(* Logix 5000 project; controller Lab1 vendor 1 type 14 code 150 rev 37.11; software revision 37.00 *)

TASK MainTask (continuous, watchdog 500 ms) : MainProgram

MODULES
   Local : vendor 1 type 14 code 150 (Compact 0, rev 37.11)
      Discrete_IO : Embedded (Compact 1, rev 3.1, Output RPI 20 ms)
      Analog_IO : Embedded (Compact 2, rev 1.1, Output RPI 80 ms)
      Counters : Embedded (Compact 3, rev 1.1, Output RPI 20 ms)
END_MODULES

VAR_GLOBAL   (* controller tags *)
   ClosingDrain : STRING;
   CountDownSec : DINT;
   CountDownStr : STRING := '0';
   Countfor60cm : DINT := 30818;
   CurrentFillTarge_cm : REAL;
   CurrentMixTime_ms : DINT;
   CurrentPassVolume_mL : REAL;
   DefaultK_factor : REAL := 13190.0;
   Done_btn : ALIAS FOR Local:1:I.Data.1;
   DotStr : STRING := '.';
   DotZeroStr : STRING := '.0';
   Drain_btn : ALIAS FOR Local:1:I.Data.3;
   DrainDisplay_EU : REAL;
   DrainEU_Int : DINT;
   DrainEU_Str : STRING;
   DrainValve : ALIAS FOR Local:1:O.Data.10;
   Dump_btn : ALIAS FOR Local:1:I.Data.12;
   DumpEmpty_cm : REAL := 1.0;
   e : STRING;
   EmergencytimeCountdown : DINT;
   FillCM_Int : DINT;
   FillCM_Str : STRING;
   FillHeight_cm_HSC : REAL;
   FillSetPoint_cm : REAL := 30.0;
   Full : DINT := 29000;
   Full_Btn : ALIAS FOR Local:1:I.Data.15;
   Good_btn : ALIAS FOR Local:1:I.Data.0;
   Half : DINT := -128;
   Half_Btn : ALIAS FOR Local:1:I.Data.14;
   HSC1_CurrentCount : ALIAS FOR Local:3:I.Ctr0CurrentCount;
   HSC_Enable : ALIAS FOR Local:3:O.Ctr0En;
   HSC_ResetPulse : ALIAS FOR Local:3:O.Ctr0SoftPreset;
   HSCStr : STRING := '30818';
   InitDone : DINT;
   InitDoneAlready : DINT;
   K_factor : REAL := 12630.327;
   LevelMax : DINT := 12354;
   LevelMin : DINT := -30607;
   LevelRaw_0cm : DINT;
   LevelRaw_85cm : DINT;
   M_DrainClose1 : STRING := 'Pass 1 : Waiting for drain valve to close';
   M_DrainClose2 : STRING := 'Pass 2 : waiting for drain valve to close';
   M_DrainClose3 : STRING;
   M_Dump : STRING := 'Normal Dump. DP display EU =';
   M_EmerDraining : STRING;
   M_Emerg : STRING := 'Emergency Stop Pressed : Press Drain to empty and recover';
   M_EmergDraining : STRING := 'Emergency Draining, Seconds left';
   M_Emergencytime : STRING;
   M_Fill : STRING := 'Normal Fill : Estimated level from HSC = ';
   M_Idle : STRING := 'Proving Selected. Press Prove to begin or Zero to reset HSC';
   M_Kcalculated : STRING := 'K - Factor Calculated. Press Done to return to Waiting.';
   M_KCalculating : STRING := 'Calculating K-Factor from captured proving run..';
   M_Mix1 : STRING := 'Pass 1 Mixing for 3 seconds';
   M_Mix2 : STRING := 'Pass 2 mixing for 2 seconds';
   M_Mix3 : STRING := 'Pass 3 mixing for 5 seconds. Price = ';
   M_Pass1Dump : STRING;
   M_Pass1Fill : STRING := 'Pass 1 filling to 30cm. Height cm =';
   M_Pass2 : STRING := 'Pass 2 preparation: resetting HSC and loading second targer';
   M_Pass2Dump : STRING := 'Pass 2 dumping. Batch finishing';
   M_Pass2Fill : STRING := 'Pass 2 filling to 20 cm. Height cm = ';
   M_Pass3Dump : STRING := 'Pass 3 dumping. Final Price = ';
   M_Pass3Fill : STRING := 'Pass 3 Filling to 50 cm. Height = ';
   M_price : STRING := '   Price in dollars = ';
   M_Proving : STRING := 'Proving: Fill. Press Good @ 60 cm , HSC  = ';
   M_Proving_Closing : STRING := 'Proving: Waiting for drain to close. Second left =';
   M_Proving_Starting : STRING := 'Proving setup: capturing low level and closing drain.';
   M_RevDrainClose1 : STRING := 'Reverse Drain Closing 1';
   M_RevDrainClose2 : STRING := 'Reverse Drain Closing 2';
   M_RevDump1 : STRING := 'Reverse Dump 1 EU';
   M_RevDump2 : STRING := 'Reverse Dump 2 EU';
   M_RevFill1 : STRING := 'Reverse Fill 1 cm';
   M_RevFill2 : STRING := 'Reverse Fill 2 cm';
   M_RevMix1 : STRING := 'Reverse Mix 1';
   M_RevMix2 : STRING := 'Reverse Mix 2';
   m_state3 : STRING;
   M_StopDump : STRING := 'Stop Dump actice. DP Display EU = ';
   M_StopHold : STRING := 'Stopped. Press Dump to empty tank and reset displayed volume.';
   M_TotalmL : STRING := 'Total Volume mL = ';
   M_Waiting2 : STRING := 'Waiting: Press Start, Reverse, or Prove';
   MaxTime_ms : DINT;
   Mixer : ALIAS FOR Local:1:O.Data.9;
   MixTimeCalc_ms : DINT;
   PassFillBase_mL : REAL;
   PassNumber : DINT;
   PressureRaw : ALIAS FOR Local:2:I.Ch3Data;
   Price_dollars : REAL;
   Price_Int : DINT;
   Price_Str : STRING;
   PriceCent_Int : DINT;
   PriceCent_Str : STRING;
   PriceDollar_Int : DINT;
   PriceDollar_Str : STRING;
   PROVE_btn : ALIAS FOR Local:1:I.Data.8;
   Pump : ALIAS FOR Local:1:O.Data.8;
   Quarter : DINT := -15000;
   Quarter_Btn : ALIAS FOR Local:1:I.Data.13;
   Raw_5cm : DINT;
   Reverse_btn : ALIAS FOR Local:1:I.Data.2;
   Seq1 : DINT;
   Seq2 : DINT := 1;
   Start_btn : ALIAS FOR Local:1:I.Data.11;
   Status : STRING := 'Press Prove to Start';
   Stop_btn : ALIAS FOR Local:1:I.Data.9;
   T_DrainClose : TIMER := (PRE := 15000);
   T_DrainClosePass1 : TIMER := (PRE := 15000);
   T_DrainClosePass2 : TIMER := (PRE := 15000);
   T_DrainClosePass3 : TIMER := (PRE := 15000);
   T_DumpPass1 : TIMER := (PRE := 15000);
   T_DumpPass2 : TIMER := (PRE := 3000);
   T_DumpPass3 : TIMER := (PRE := 15000);
   T_EmergencyDrain : TIMER := (PRE := 15000);
   T_InitHold : TIMER := (PRE := 1000);
   T_Mix : TIMER;
   T_NormalDump : TIMER := (PRE := 3000);
   T_StopDump : TIMER := (PRE := 30000);
   TankLevel_cm : REAL;
   TankLevelRaw : ALIAS FOR Local:2:I.Ch3Data;
   TargetTicks : REAL;
   TargetTicks90 : REAL;
   TempStr : STRING;
   TotalVolume_mL : REAL;
   ValveClosed : DINT := -32767;
   ValveOpen : DINT := 29000;
   ValvePosition : ALIAS FOR Local:2:O.Ch1Data;
   Volume_mL_Int : DINT;
   Volume_mL_Str : STRING;
   Zero_btn : ALIAS FOR Local:1:I.Data.10;
END_VAR

PROGRAM MainProgram   (* main routine MainRoutine *)
VAR
   DumpEmptyRev_cm : REAL := 0.02;
   Pricee : STRING := 'The Price (in dollars) =  ';
   T_DrainCloseRev1 : TIMER := (PRE := 15000);
   T_DrainCloseRev2 : TIMER := (PRE := 15000);
   T_RevDump1 : TIMER := (PRE := 15000);
   T_RevDump2 : TIMER := (PRE := 15000);
   T_RevEmptyConfirm : TIMER := (PRE := 1000);
   T_RevEmptyConfirm2 : TIMER := (PRE := 1000);
END_VAR

ROUTINE _m   (* structured text *)
   Price_Int := (Price_dollars * 100.0) + 0.5;
   PriceDollar_Int := Price_Int / 100;
   PriceCent_Int := Price_Int MOD 100;
   
   DTOS(PriceDollar_Int, PriceDollar_Str);
   DTOS(PriceCent_Int, PriceCent_Str);
   
   if(PriceCent_Int < 10) then
   	CONCAT(PriceDollar_Str, DotZeroStr,TempStr);
   else
   	CONCAT(PriceDollar_Str, DotStr, TempStr);
   end_if;
   
   CONCAT(TempStr, PriceCent_Str, Price_Str);
   
   if Seq2 = 1 then
   	Concat(M_Idle, e, Status);
   
   elsif Seq2 = 2 then
   	CONCAT(M_Proving_Starting,e,Status);
   
   elsif Seq2 = 3 then
   	CountDownSec:= (T_DrainClose.PRE - T_DrainClose.ACC)/1000;
   	DTOS(CountDownSec,CountDownStr);
   	CONCAT(M_Proving_Closing, CountDownStr,Status);
   
   ElSIF Seq2 = 4 then
   	DTOS(HSC1_CurrentCount,HSCStr);
   	CONCAT(M_Proving, HSCStr,Status);
   
   Elsif Seq2 = 5 then
   	CONCAT(M_KCalculating, e,Status);
   
   elsif Seq2 = 6 then
   	CONCAT(M_Kcalculated, e ,Status);
   
   elsif Seq2 = 90 then
   	CONCAT(M_Emerg,e,Status);
   
   Elsif Seq2 = 91 then
   	EmergencytimeCountdown:= (T_EmergencyDrain.PRE-T_EmergencyDrain.ACC)/1000;
   	DTOS(EmergencytimeCountdown, M_Emergencytime);
   	CONCAT(M_EmerDraining,M_Emergencytime, Status);
   
   elsif Seq1 = 2 then
   	CONCAT(M_Waiting2,e,Status);
   
   elsif
   	Seq1 = 3 then
   	FillCM_Int:= FillHeight_cm_HSC + 0.999;
   	DTOS(FillCM_Int,FillCM_Str);
   	Volume_mL_Int:= TotalVolume_mL+0.5;
   	DTOS(Volume_mL_Int, Volume_mL_Str);
   	CONCAT(M_Pass1Fill,FillCM_Str,Status);
   	CONCAT(Status, M_TotalmL, Status);
   	CONCAT(Status,Volume_mL_Str,Status);
   
   elsif Seq1 = 4 then
   	CONCAT(M_Mix1,e,Status);
   
   elsif Seq1 = 5 then
   	DrainEU_Int:=DrainDisplay_EU + 0.5;
   	DTOS(DrainEU_Int, DrainEU_Str);
   	CONCAT(M_Pass1Dump, DrainEU_Str,Status);
   
   elsif Seq1 = 6 then
   	CONCAT(M_StopHold,e,Status);
   
   elsif Seq1 = 7 then
   	DrainEU_Int:=DrainDisplay_EU + 0.5;
   	DTOS(DrainEU_Int, DrainEU_Str);
   	CONCAT(M_StopDump,DrainEU_Str,Status);
   
   elsif Seq1 = 8 then
   	CountDownSec := (T_DrainClosePass2.PRE - T_DrainClosePass2.ACC) / 1000;
   	DTOS(CountDownSec, CountDownStr);
   	CONCAT(M_DrainClose2, CountDownStr, Status);
   
   elsif Seq1 = 9 then
   	FillCM_Int:= FillHeight_cm_HSC + 0.999;
   	DTOS(FillCM_Int, FillCM_Str);
   
   	Volume_mL_Int:= TotalVolume_mL + 0.5;
   	DTOS(Volume_mL_Int, Volume_mL_Str);
   	CONCAT(M_Pass2Fill, FillCM_Str,Status);
   
   	concat(Status,M_TotalmL,Status);
   	CONCAT(Status, Volume_mL_Str, Status);
   
   elsif Seq1 = 10 then
   	CONCAT(M_Mix2, e,Status);
   
   elsif Seq1 = 11 then
   	DrainEU_Int:=DrainDisplay_EU + 0.5;
   	DTOS(DrainEU_Int, DrainEU_Str);
   	CONCAT(M_Pass2Dump,DrainEU_Str,Status);
   
   elsif Seq1 = 12 then
   	CountDownSec := (T_DrainClosePass1.PRE - T_DrainClosePass1.ACC) / 1000;
   	DTOS(CountDownSec, CountDownStr);
   	CONCAT(M_DrainClose1,CountDownStr,Status);
   
   elsif Seq1 = 13 then
   	CountDownSec := (T_DrainClosePass3.PRE - T_DrainClosePass3.ACC) / 1000;
   	DTOS(CountDownSec, CountDownStr);
   	CONCAT(M_DrainClose3,CountDownStr,Status);
   
   elsif Seq1 = 14 then
   	FillCM_Int := FillHeight_cm_HSC+ 0.999;
   	DTOS(FillCM_Int,FillCM_Str);
   
   	Volume_mL_Int := TotalVolume_mL + 0.5;
   	DTOS(Volume_mL_Int,Volume_mL_Str);
   
   	CONCAT(M_Pass3Fill, FillCM_Str, Status);
   	CONCAT(Status, M_TotalmL, Status);
   	CONCAT(Status, Volume_mL_Str, Status);
   	CONCAT(Status, M_price,Status);
   	CONCAT(Status, Price_Str, Status);
   
   elsif Seq1 = 15 then
   	CONCAT(M_Mix3, M_price, Status);
   	CONCAT(Status, Price_Str, Status);
   
   elsif Seq1 = 16 then
   
   	DrainEU_Int:=DrainDisplay_EU + 0.5;
   	DTOS(DrainEU_Int, DrainEU_Str);
   
   	Concat(M_Pass3Dump, DrainEU_Str, Status);
   	CONCAT(Status, M_price, Status);
   	CONCAT(Status, Price_Str,Status);
   
   
   elsif Seq1 = 17 then
   	Concat(M_RevMix1,e,Status);
   
   elsif Seq1 = 18 then
   
   	Concat(M_RevDrainClose1,e,Status);
   
   elsif Seq1 = 19 then
   	FillCM_Int := FillHeight_cm_HSC + 0.999;
   	DTOS(FillCM_Int, FillCM_Str);
   	Concat(M_RevFill1,FillCM_Str,Status);
   
   elsif Seq1 = 20 then
   	DrainEU_Int:= DrainDisplay_EU + 0.5;
   	DTOS(DrainEU_Int, DrainEU_Str);
   	CONCAT(M_RevDump1,DrainEU_Str,Status);
   
   elsif Seq1 = 21 then
   	CONCAT(M_RevMix2,e,Status);
   
   elsif Seq1 = 22 then
   	Concat(M_RevDrainClose2,e,Status);
   
   elsif Seq1 = 23 then
   	FillCM_Int := FillHeight_cm_HSC + 0.999;
   	DTOS(FillCM_Int, FillCM_Str);
   	Concat(M_RevFill2,FillCM_Str,Status);
   
   elsif Seq1 = 24 then
   	DrainEU_Int:= DrainDisplay_EU + 0.5;
   	DTOS(DrainEU_Int, DrainEU_Str);
   	CONCAT(M_RevDump2,DrainEU_Str,Status);
   
   end_if;
   
END_ROUTINE

ROUTINE MainRoutine   (* ladder *)
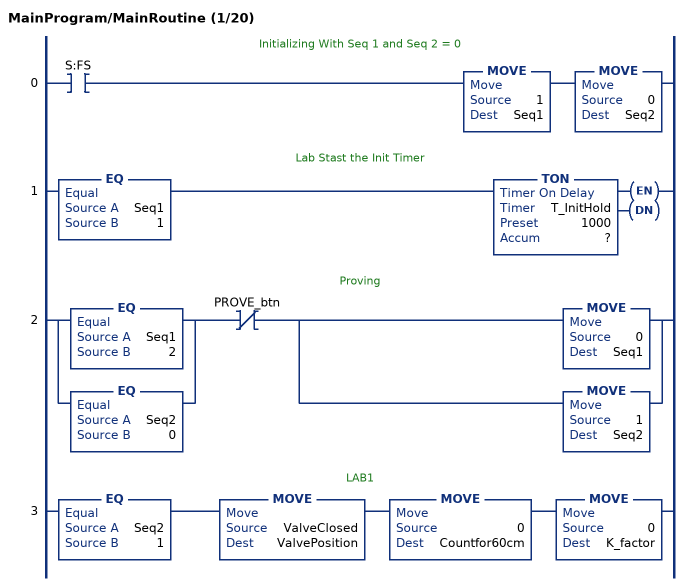
   // Initializing With Seq 1 and Seq 2 = 0
   0: XIC(S:FS)MOVE(1,Seq1)MOVE(0,Seq2);
   // Lab Stast the Init Timer
   1: EQ(Seq1,1)TON(T_InitHold,?,?);
   // Proving
   2: [EQ(Seq1,2) ,EQ(Seq2,0) ]XIO(PROVE_btn)[MOVE(0,Seq1) ,MOVE(1,Seq2) ];
   // LAB1
   3: EQ(Seq2,1)MOVE(ValveClosed,ValvePosition)MOVE(0,Countfor60cm)MOVE(0,K_factor);
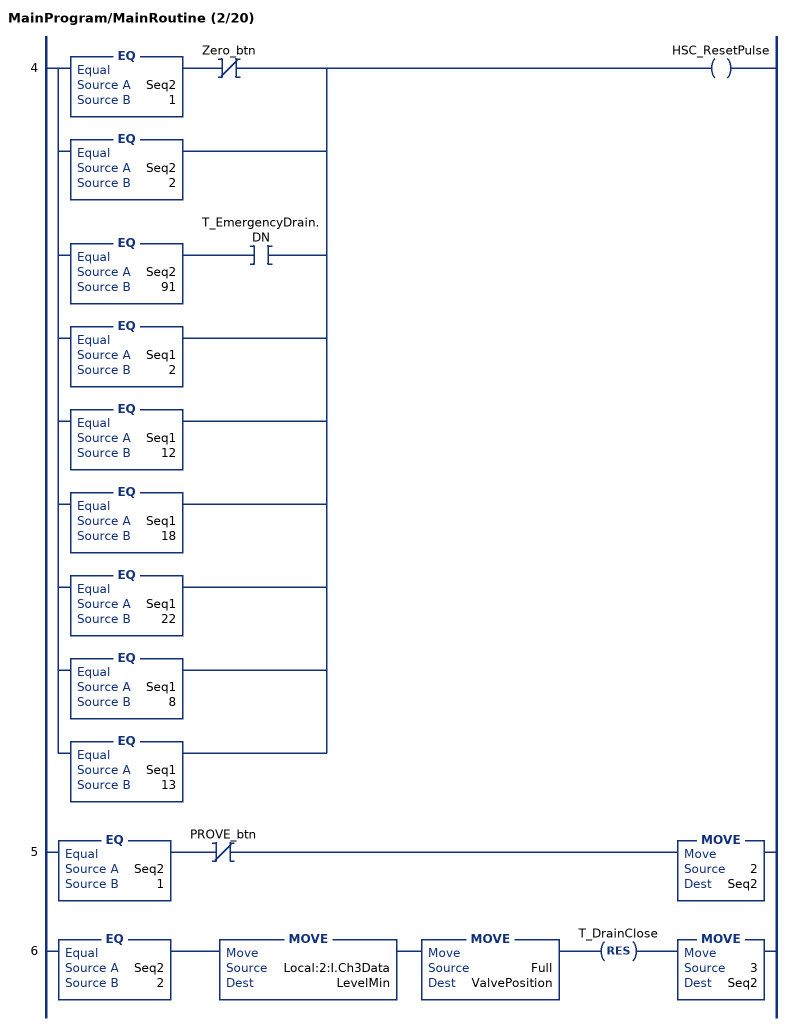
   4: [EQ(Seq2,1) XIO(Zero_btn) ,[EQ(Seq2,2) ,[EQ(Seq2,91) XIC(T_EmergencyDrain.DN) ,EQ(Seq1,2) ,EQ(Seq1,12) ,EQ(Seq1,18) ,EQ(Seq1,22) ,EQ(Seq1,8) ,EQ(Seq1,13) ] ] ]OTE(HSC_ResetPulse);
   5: EQ(Seq2,1)XIO(PROVE_btn)MOVE(2,Seq2);
   6: EQ(Seq2,2)MOVE(Local:2:I.Ch3Data,LevelMin)MOVE(Full,ValvePosition)RES(T_DrainClose)MOVE(3,Seq2);
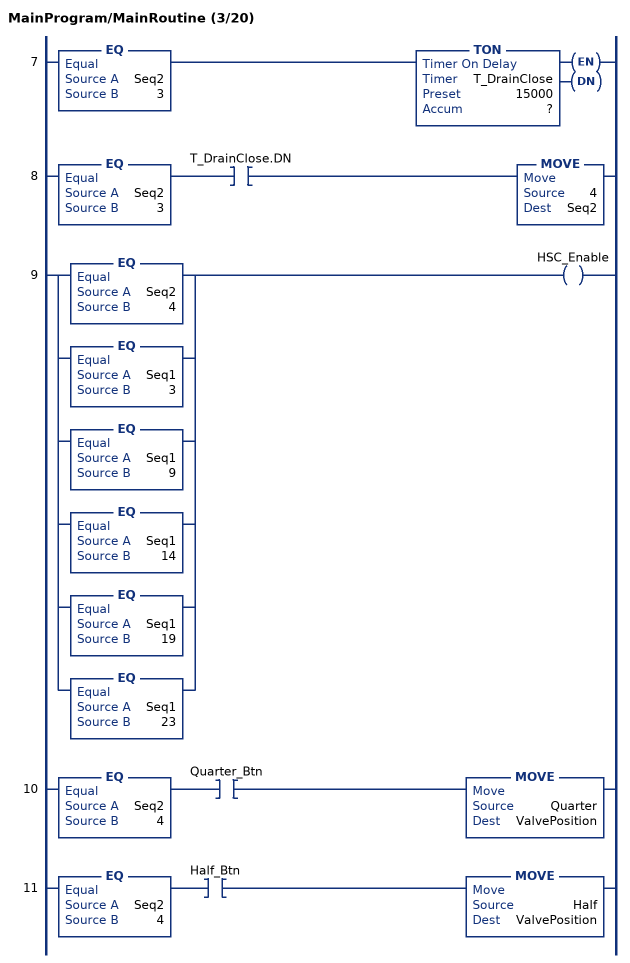
   7: EQ(Seq2,3)TON(T_DrainClose,?,?);
   8: EQ(Seq2,3)XIC(T_DrainClose.DN)MOVE(4,Seq2);
   9: [EQ(Seq2,4) ,[EQ(Seq1,3) ,[EQ(Seq1,9) ,EQ(Seq1,14) ,EQ(Seq1,19) ,EQ(Seq1,23) ] ] ]OTE(HSC_Enable);
   10: EQ(Seq2,4)XIC(Quarter_Btn)MOVE(Quarter,ValvePosition);
   11: EQ(Seq2,4)XIC(Half_Btn)MOVE(Half,ValvePosition);
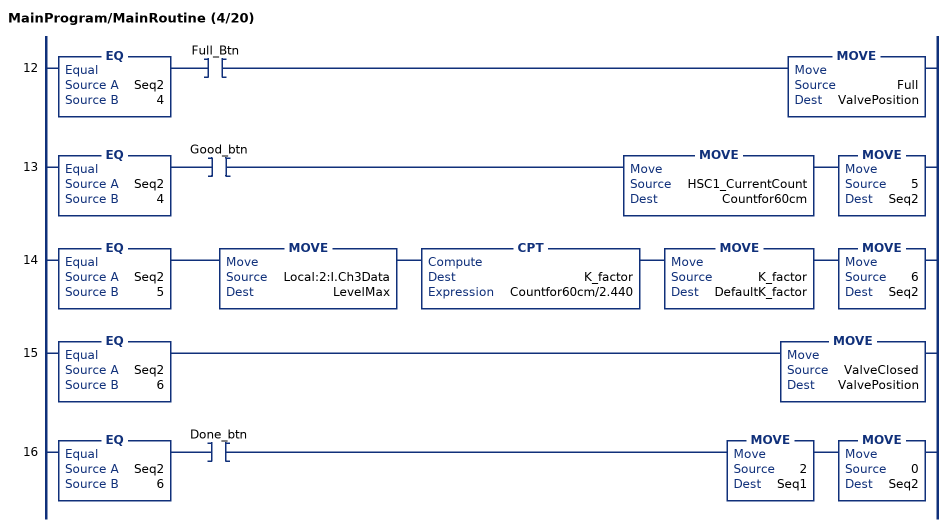
   12: EQ(Seq2,4)XIC(Full_Btn)MOVE(Full,ValvePosition);
   13: EQ(Seq2,4)XIC(Good_btn)MOVE(HSC1_CurrentCount,Countfor60cm)MOVE(5,Seq2);
   14: EQ(Seq2,5)MOVE(Local:2:I.Ch3Data,LevelMax)CPT(K_factor,Countfor60cm/2.440)MOVE(K_factor,DefaultK_factor)MOVE(6,Seq2);
   15: EQ(Seq2,6)MOVE(ValveClosed,ValvePosition);
   16: EQ(Seq2,6)XIC(Done_btn)MOVE(2,Seq1)MOVE(0,Seq2);
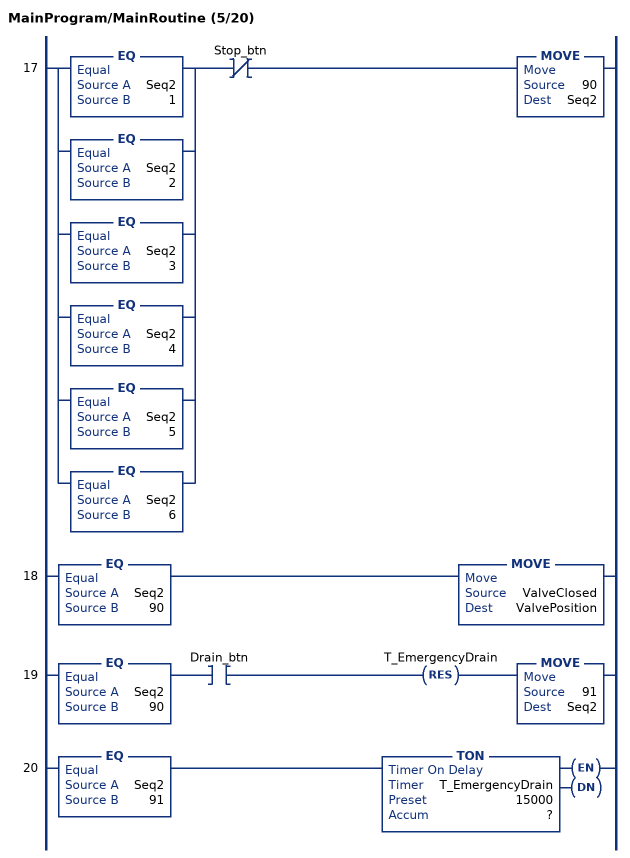
   17: [EQ(Seq2,1) ,[EQ(Seq2,2) ,[EQ(Seq2,3) ,[EQ(Seq2,4) ,[EQ(Seq2,5) ,EQ(Seq2,6) ] ] ] ] ]XIO(Stop_btn)MOVE(90,Seq2);
   18: EQ(Seq2,90)MOVE(ValveClosed,ValvePosition);
   19: EQ(Seq2,90)XIC(Drain_btn)RES(T_EmergencyDrain)MOVE(91,Seq2);
   20: EQ(Seq2,91)TON(T_EmergencyDrain,?,?);
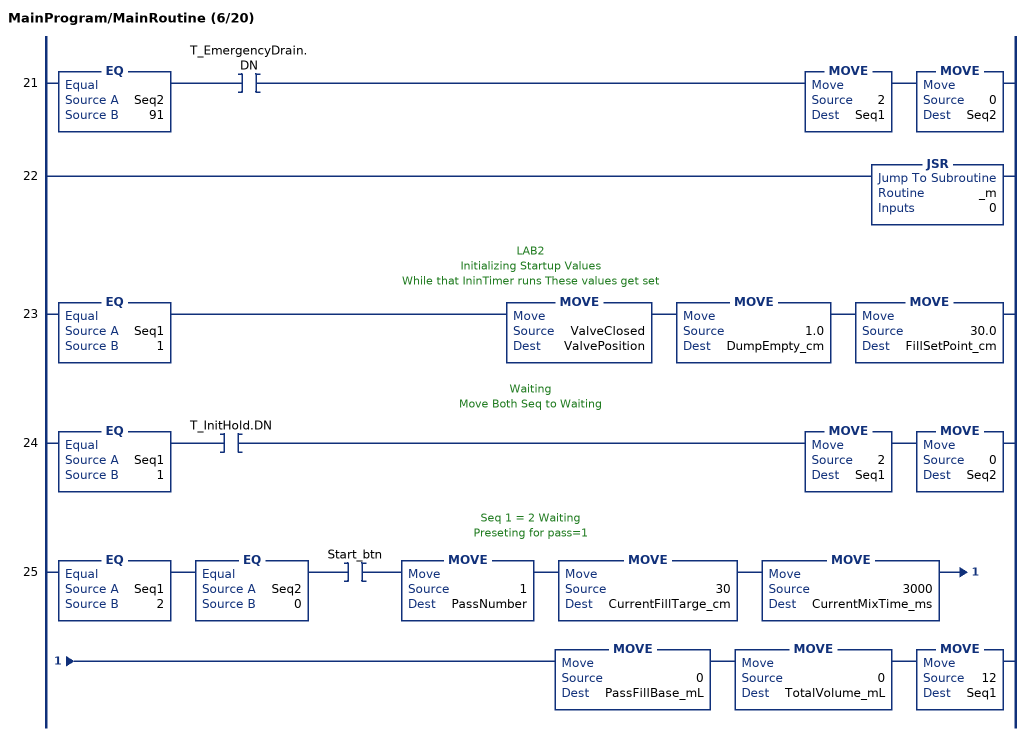
   21: EQ(Seq2,91)XIC(T_EmergencyDrain.DN)MOVE(2,Seq1)MOVE(0,Seq2);
   22: JSR(_m,0);
   // LAB2
   // Initializing Startup Values
   // While that IninTimer runs These values get set
   23: EQ(Seq1,1)MOVE(ValveClosed,ValvePosition)MOVE(1.0,DumpEmpty_cm)MOVE(30.0,FillSetPoint_cm);
   // Waiting
   // Move Both Seq to Waiting
   24: EQ(Seq1,1)XIC(T_InitHold.DN)MOVE(2,Seq1)MOVE(0,Seq2);
   // Seq 1 = 2 Waiting
   // Preseting for pass=1
   25: EQ(Seq1,2)EQ(Seq2,0)XIC(Start_btn)MOVE(1,PassNumber)MOVE(30,CurrentFillTarge_cm)MOVE(3000,CurrentMixTime_ms)MOVE(0,PassFillBase_mL)MOVE(0,TotalVolume_mL)MOVE(12,Seq1);
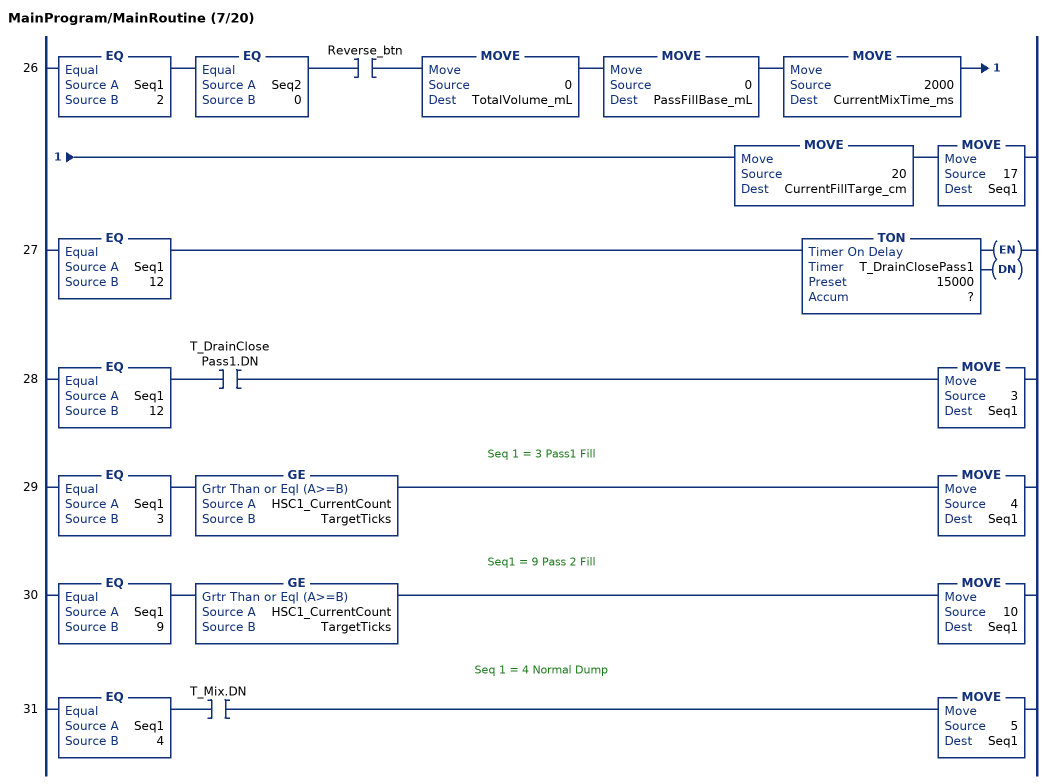
   26: EQ(Seq1,2)EQ(Seq2,0)XIC(Reverse_btn)MOVE(0,TotalVolume_mL)MOVE(0,PassFillBase_mL)MOVE(2000,CurrentMixTime_ms)MOVE(20,CurrentFillTarge_cm)MOVE(17,Seq1);
   27: EQ(Seq1,12)TON(T_DrainClosePass1,?,?);
   28: EQ(Seq1,12)XIC(T_DrainClosePass1.DN)MOVE(3,Seq1);
   // Seq 1 = 3 Pass1 Fill
   29: EQ(Seq1,3)GE(HSC1_CurrentCount,TargetTicks)MOVE(4,Seq1);
   // Seq1 = 9 Pass 2 Fill
   30: EQ(Seq1,9)GE(HSC1_CurrentCount,TargetTicks)MOVE(10,Seq1);
   // Seq 1 = 4 Normal Dump
   31: EQ(Seq1,4)XIC(T_Mix.DN)MOVE(5,Seq1);
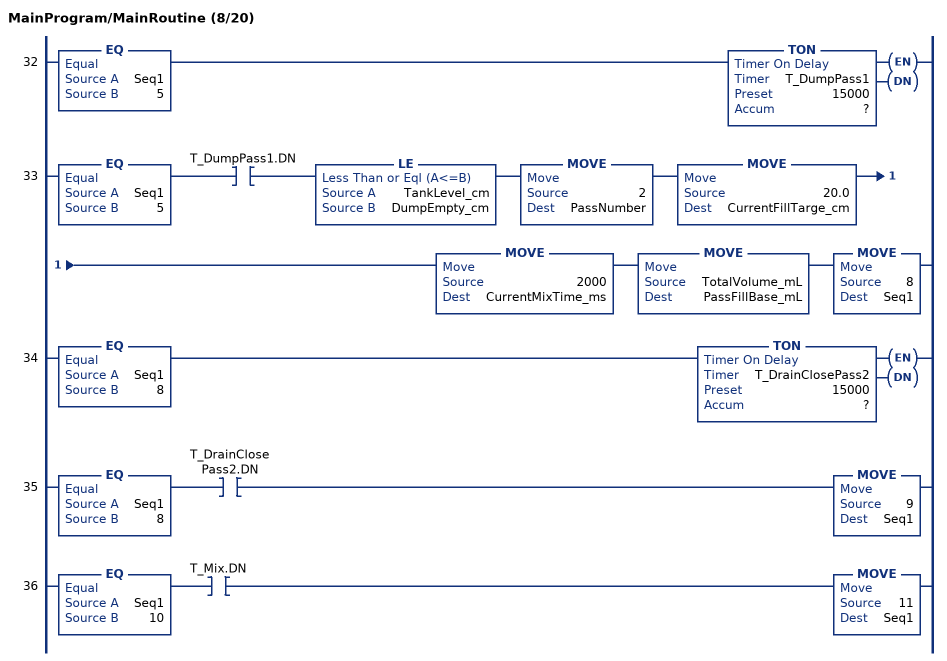
   32: EQ(Seq1,5)TON(T_DumpPass1,?,?);
   33: EQ(Seq1,5)XIC(T_DumpPass1.DN)LE(TankLevel_cm,DumpEmpty_cm)MOVE(2,PassNumber)MOVE(20.0,CurrentFillTarge_cm)MOVE(2000,CurrentMixTime_ms)MOVE(TotalVolume_mL,PassFillBase_mL)MOVE(8,Seq1);
   34: EQ(Seq1,8)TON(T_DrainClosePass2,?,?);
   35: EQ(Seq1,8)XIC(T_DrainClosePass2.DN)MOVE(9,Seq1);
   36: EQ(Seq1,10)XIC(T_Mix.DN)MOVE(11,Seq1);
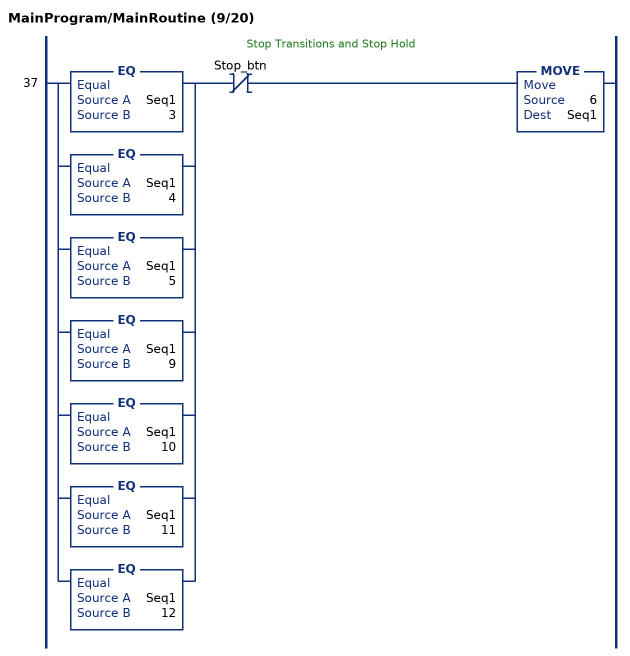
   // Stop Transitions and Stop Hold
   37: [EQ(Seq1,3) ,[EQ(Seq1,4) ,[EQ(Seq1,5) ,[EQ(Seq1,9) ,[EQ(Seq1,10) ,[EQ(Seq1,11) ,EQ(Seq1,12) ] ] ] ] ] ]XIO(Stop_btn)MOVE(6,Seq1);
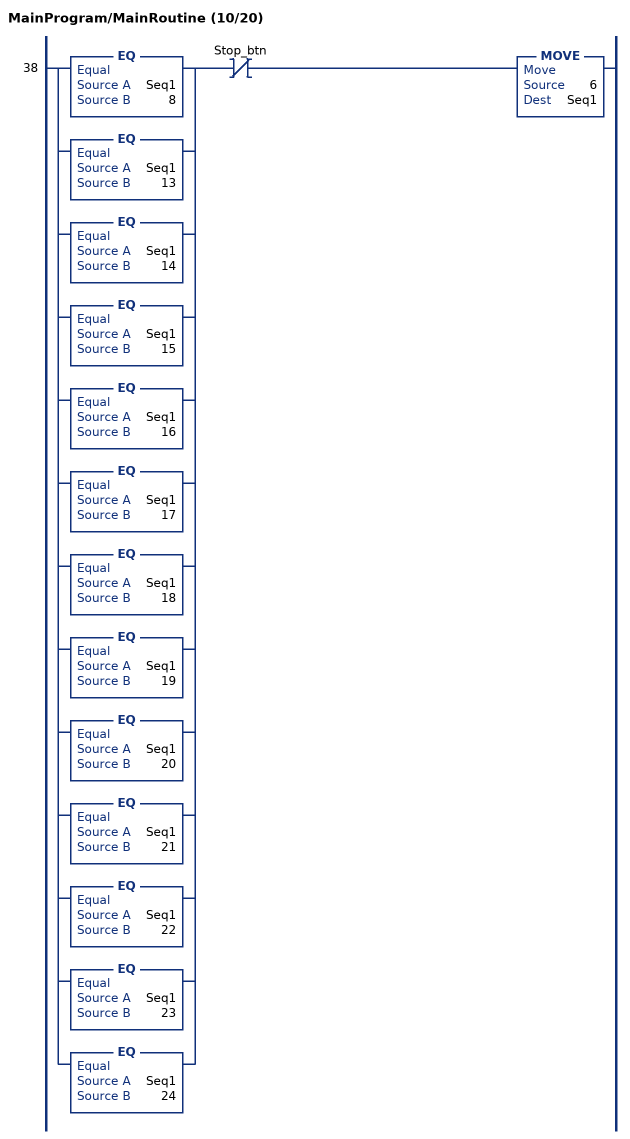
   38: [EQ(Seq1,8) ,[EQ(Seq1,13) ,[EQ(Seq1,14) ,[EQ(Seq1,15) ,EQ(Seq1,16) ,EQ(Seq1,17) ,EQ(Seq1,18) ,EQ(Seq1,19) ,EQ(Seq1,20) ,EQ(Seq1,21) ,EQ(Seq1,22) ,EQ(Seq1,23) ,EQ(Seq1,24) ] ] ] ]XIO(Stop_btn)MOVE(6,Seq1);
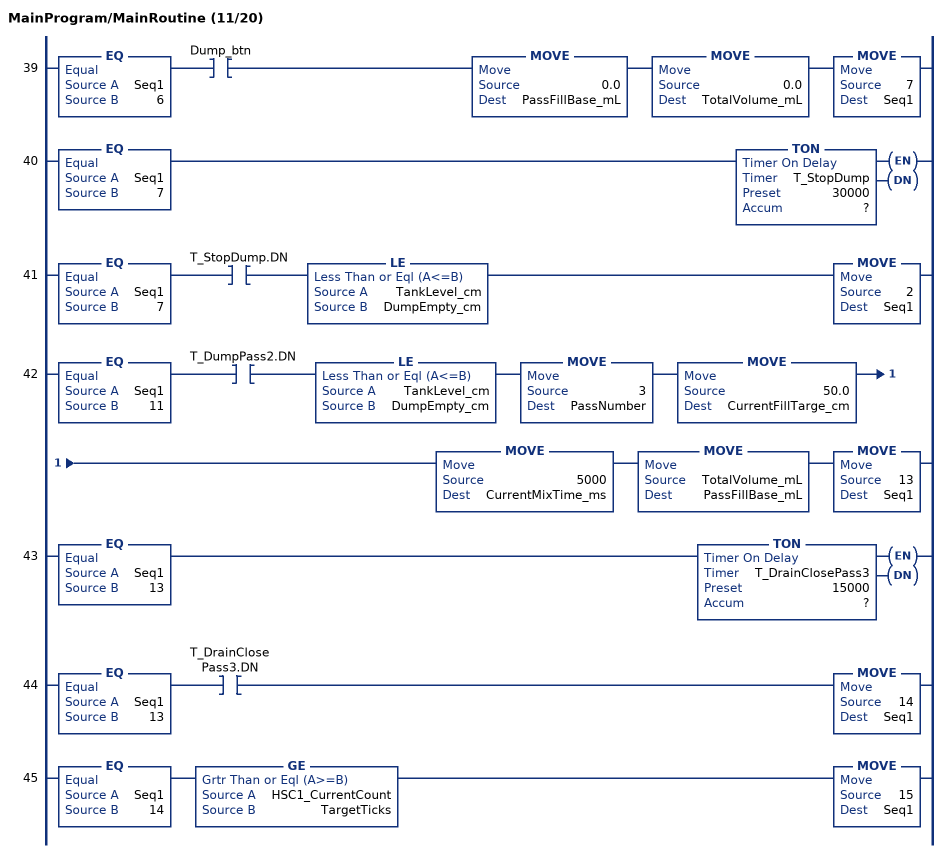
   39: EQ(Seq1,6)XIC(Dump_btn)MOVE(0.0,PassFillBase_mL)MOVE(0.0,TotalVolume_mL)MOVE(7,Seq1);
   40: EQ(Seq1,7)TON(T_StopDump,?,?);
   41: EQ(Seq1,7)XIC(T_StopDump.DN)LE(TankLevel_cm,DumpEmpty_cm)MOVE(2,Seq1);
   42: EQ(Seq1,11)XIC(T_DumpPass2.DN)LE(TankLevel_cm,DumpEmpty_cm)MOVE(3,PassNumber)MOVE(50.0,CurrentFillTarge_cm)MOVE(5000,CurrentMixTime_ms)MOVE(TotalVolume_mL,PassFillBase_mL)MOVE(13,Seq1);
   43: EQ(Seq1,13)TON(T_DrainClosePass3,?,?);
   44: EQ(Seq1,13)XIC(T_DrainClosePass3.DN)MOVE(14,Seq1);
   45: EQ(Seq1,14)GE(HSC1_CurrentCount,TargetTicks)MOVE(15,Seq1);
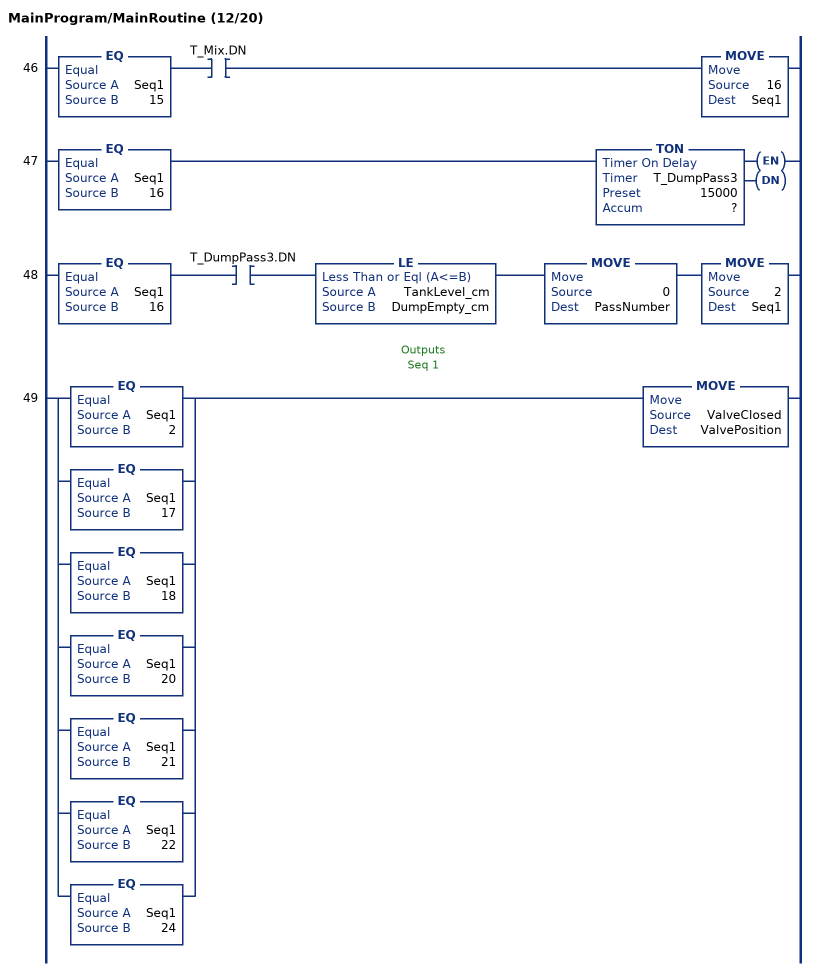
   46: EQ(Seq1,15)XIC(T_Mix.DN)MOVE(16,Seq1);
   47: EQ(Seq1,16)TON(T_DumpPass3,?,?);
   48: EQ(Seq1,16)XIC(T_DumpPass3.DN)LE(TankLevel_cm,DumpEmpty_cm)MOVE(0,PassNumber)MOVE(2,Seq1);
   // Outputs
   // Seq 1
   49: [EQ(Seq1,2) ,EQ(Seq1,17) ,EQ(Seq1,18) ,EQ(Seq1,20) ,EQ(Seq1,21) ,EQ(Seq1,22) ,EQ(Seq1,24) ]MOVE(ValveClosed,ValvePosition);
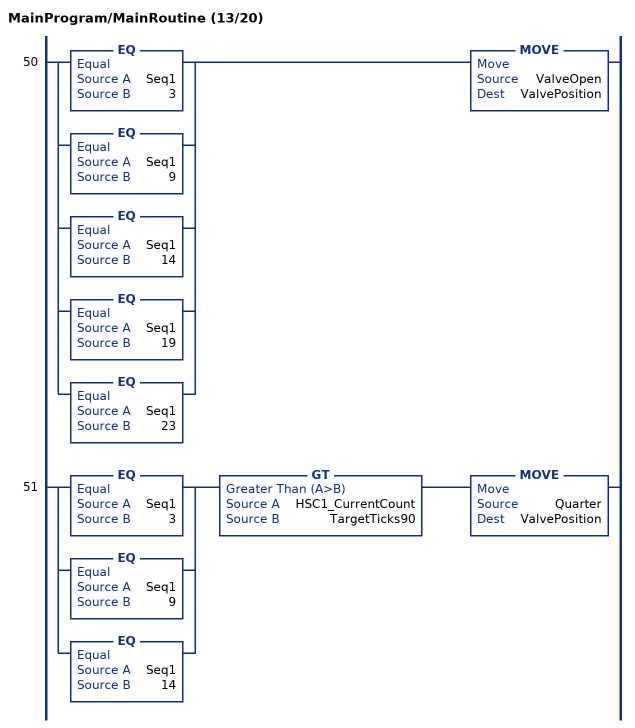
   50: [EQ(Seq1,3) ,[EQ(Seq1,9) ,EQ(Seq1,14) ,EQ(Seq1,19) ,EQ(Seq1,23) ] ]MOVE(ValveOpen,ValvePosition);
   51: [EQ(Seq1,3) ,[EQ(Seq1,9) ,EQ(Seq1,14) ] ]GT(HSC1_CurrentCount,TargetTicks90)MOVE(Quarter,ValvePosition);
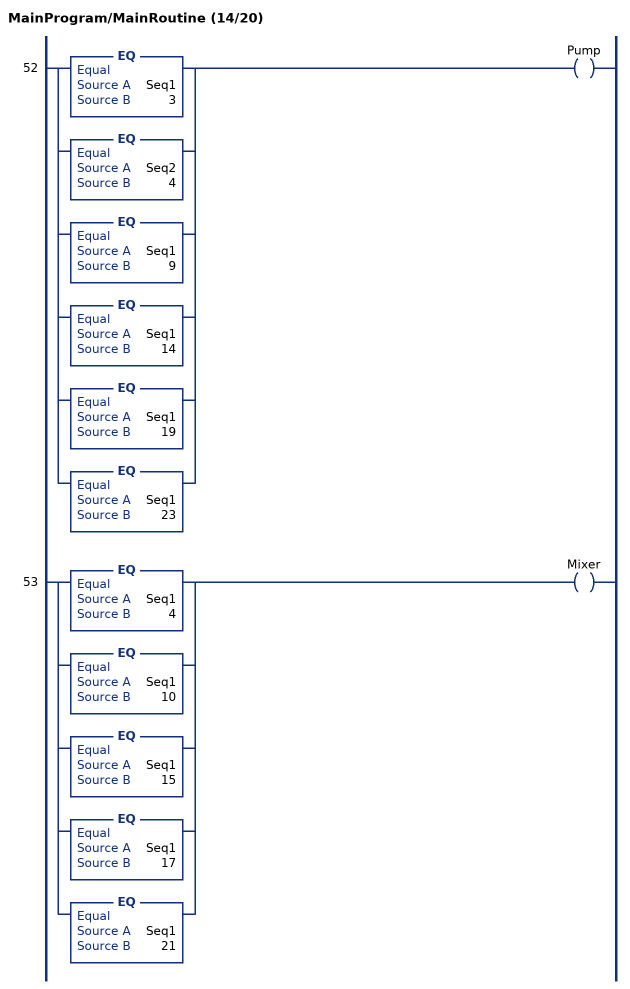
   52: [EQ(Seq1,3) ,[EQ(Seq2,4) ,[EQ(Seq1,9) ,[EQ(Seq1,14) ,EQ(Seq1,19) ,EQ(Seq1,23) ] ] ] ]OTE(Pump);
   53: [EQ(Seq1,4) ,[EQ(Seq1,10) ,EQ(Seq1,15) ,EQ(Seq1,17) ,EQ(Seq1,21) ] ]OTE(Mixer);
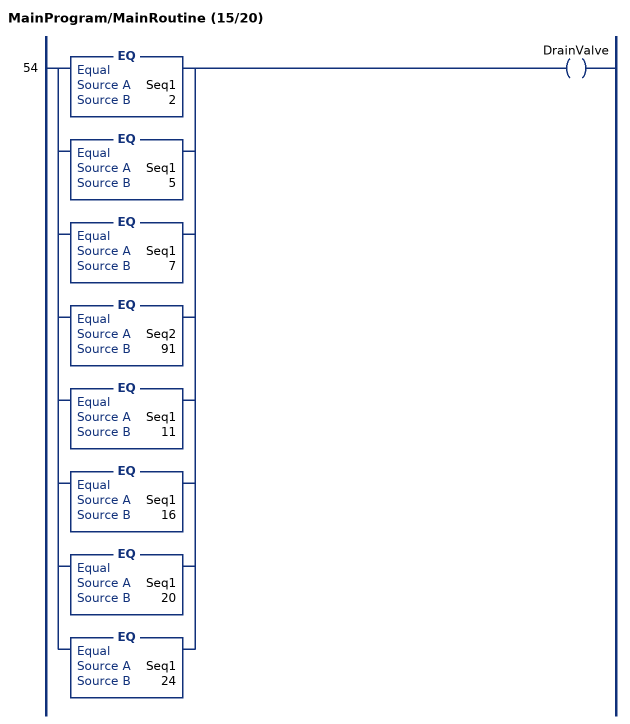
   54: [EQ(Seq1,2) ,[EQ(Seq1,5) ,[EQ(Seq1,7) ,[EQ(Seq2,91) ,[EQ(Seq1,11) ,[EQ(Seq1,16) ,EQ(Seq1,20) ,EQ(Seq1,24) ] ] ] ] ] ]OTE(DrainValve);
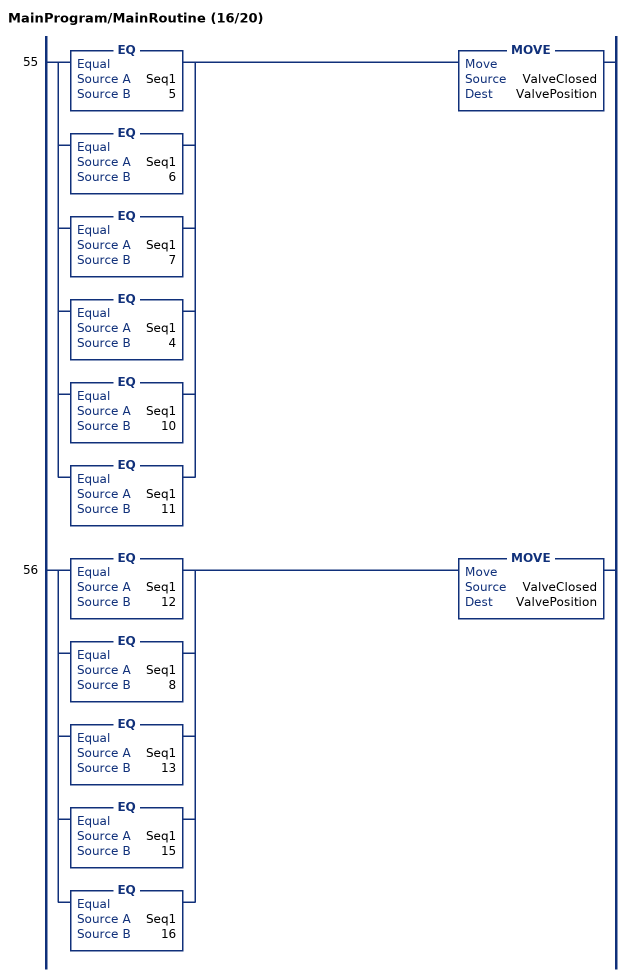
   55: [EQ(Seq1,5) ,[EQ(Seq1,6) ,[EQ(Seq1,7) ,[EQ(Seq1,4) ,[EQ(Seq1,10) ,EQ(Seq1,11) ] ] ] ] ]MOVE(ValveClosed,ValvePosition);
   56: [EQ(Seq1,12) ,[EQ(Seq1,8) ,[EQ(Seq1,13) ,[EQ(Seq1,15) ,EQ(Seq1,16) ] ] ] ]MOVE(ValveClosed,ValvePosition);
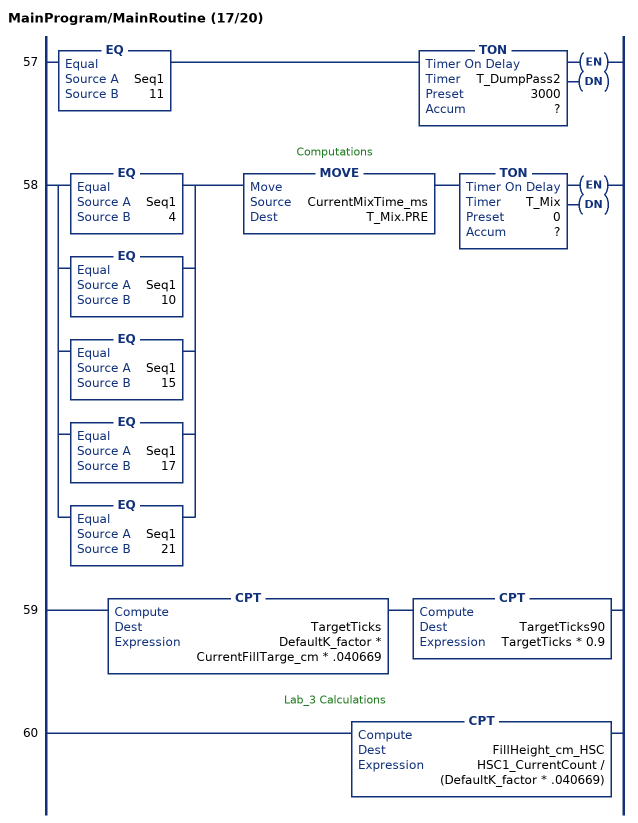
   57: EQ(Seq1,11)TON(T_DumpPass2,?,?);
   // Computations
   58: [EQ(Seq1,4) ,[EQ(Seq1,10) ,[EQ(Seq1,15) ,EQ(Seq1,17) ,EQ(Seq1,21) ] ] ]MOVE(CurrentMixTime_ms,T_Mix.PRE)TON(T_Mix,?,?);
   59: CPT(TargetTicks,DefaultK_factor * CurrentFillTarge_cm * .040669)CPT(TargetTicks90,TargetTicks * 0.9);
   // Lab_3 Calculations
   60: CPT(FillHeight_cm_HSC,HSC1_CurrentCount / (DefaultK_factor * .040669));
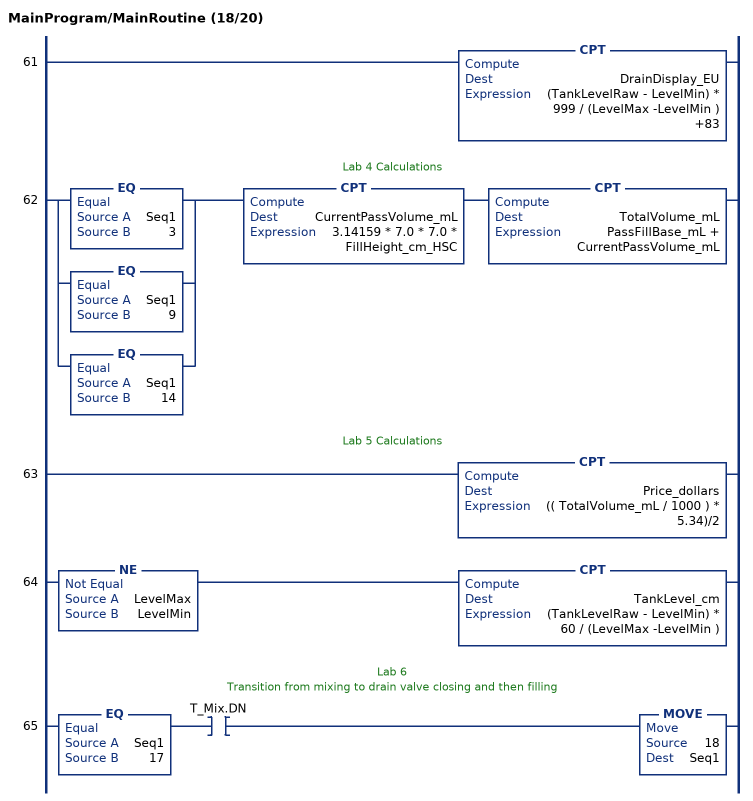
   61: CPT(DrainDisplay_EU,(TankLevelRaw - LevelMin) * 999 / (LevelMax -LevelMin ) +83);
   // Lab 4 Calculations
   62: [EQ(Seq1,3) ,[EQ(Seq1,9) ,EQ(Seq1,14) ] ]CPT(CurrentPassVolume_mL,3.14159 * 7.0 * 7.0 * FillHeight_cm_HSC)CPT(TotalVolume_mL,PassFillBase_mL + CurrentPassVolume_mL);
   // Lab 5 Calculations
   63: CPT(Price_dollars,(( TotalVolume_mL / 1000 ) * 5.34)/2);
   64: NE(LevelMax,LevelMin)CPT(TankLevel_cm,(TankLevelRaw - LevelMin) * 60 / (LevelMax -LevelMin ));
   // Lab 6
   // Transition from mixing to drain valve closing and then filling
   65: EQ(Seq1,17)XIC(T_Mix.DN)MOVE(18,Seq1);
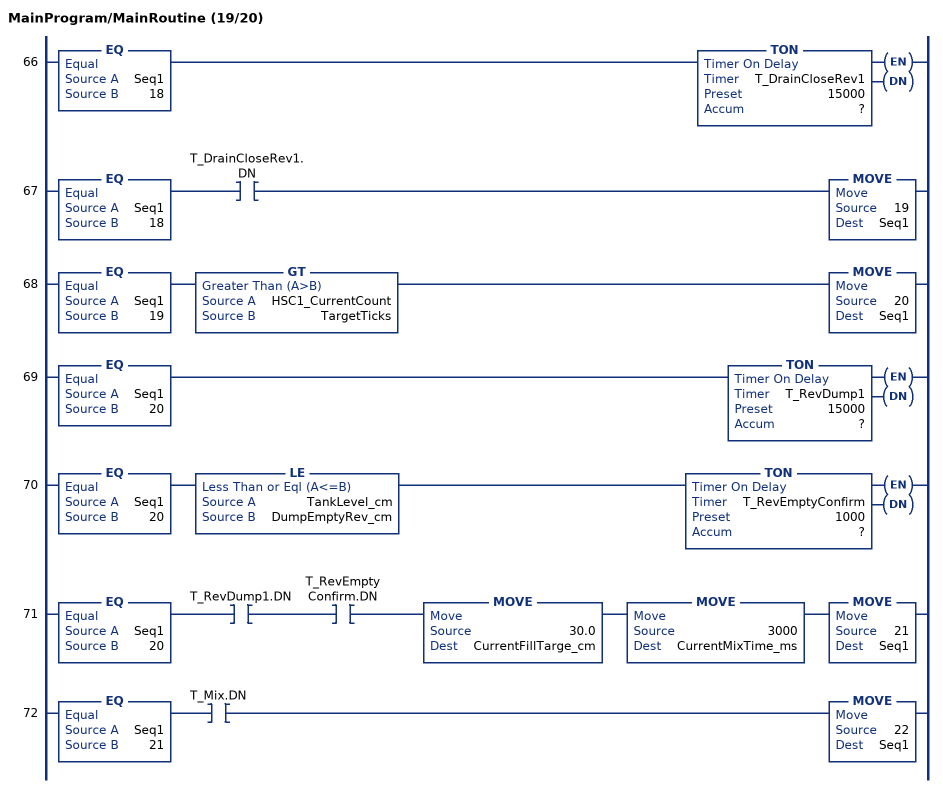
   66: EQ(Seq1,18)TON(T_DrainCloseRev1,?,?);
   67: EQ(Seq1,18)XIC(T_DrainCloseRev1.DN)MOVE(19,Seq1);
   68: EQ(Seq1,19)GT(HSC1_CurrentCount,TargetTicks)MOVE(20,Seq1);
   69: EQ(Seq1,20)TON(T_RevDump1,?,?);
   70: EQ(Seq1,20)LE(TankLevel_cm,DumpEmptyRev_cm)TON(T_RevEmptyConfirm,?,?);
   71: EQ(Seq1,20)XIC(T_RevDump1.DN)XIC(T_RevEmptyConfirm.DN)MOVE(30.0,CurrentFillTarge_cm)MOVE(3000,CurrentMixTime_ms)MOVE(21,Seq1);
   72: EQ(Seq1,21)XIC(T_Mix.DN)MOVE(22,Seq1);
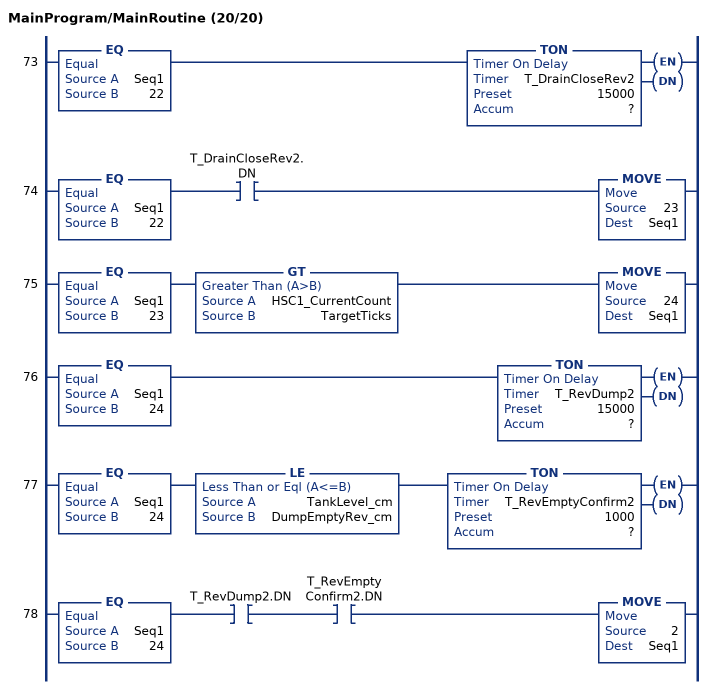
   73: EQ(Seq1,22)TON(T_DrainCloseRev2,?,?);
   74: EQ(Seq1,22)XIC(T_DrainCloseRev2.DN)MOVE(23,Seq1);
   75: EQ(Seq1,23)GT(HSC1_CurrentCount,TargetTicks)MOVE(24,Seq1);
   76: EQ(Seq1,24)TON(T_RevDump2,?,?);
   77: EQ(Seq1,24)LE(TankLevel_cm,DumpEmptyRev_cm)TON(T_RevEmptyConfirm2,?,?);
   78: EQ(Seq1,24)XIC(T_RevDump2.DN)XIC(T_RevEmptyConfirm2.DN)MOVE(2,Seq1);
END_ROUTINE
END_PROGRAM
